Yaskawa INFORM job: TSYNC-R.JBI

/JOB
//NAME TSYNC-R
//POS
///NPOS 0,0,0,0,0,0
//INST
///DATE 2022/02/07 15:21
///ATTR SC,RW,RJ,MC
////FRAME ROBOT
///LVARS 1,0,0,0,0,0,0,0
NOP
*LABEL
PULSE OT#(1616) T=0.50
WAIT IN#(1616)=ON T=0.50
JUMP *LABEL IF IN#(1616)=OFF
TIMER T=0.10
GETARG LB000 IARG#(1)
DOUT OG#(203) LB000
WAIT IG#(203)=LB000 T=0.50
JUMP *LABEL IF IG#(203)<>LB000
TIMER T=0.20
DOUT OG#(203) 0
WAIT IG#(203)=0
TIMER T=0.10
END
